PROGRAM MAIN
VAR
END_VAR

END_PROGRAM

(* stored: Version 1.1.0.1, ProductVersion 3.1.0.36
   POU MAIN: Id {8c4c05b5-5a48-4c8e-92c9-2906737a8de2} *)
